FUNCTION_BLOCK DigitalOut
VAR_INPUT
END_VAR
VAR_OUTPUT
END_VAR
VAR
	DO_io  AT %Q*: BOOL;
	timerOn : TON;
	timerOff : TON;
	onActive : BOOL;
	offActive : BOOL;
	Do_in: BOOL;
	ActualCycle : UDINT;
	fbGetCurrTask : GETCURTASKINDEX;
	NextOn: UDINT;
	NextOff :UDINT;
	fifo : FB_Fifo;
	NextOnOff : ST_streamOutputs;
	init: BOOL;
END_VAR


IF init THEN
	init := FALSE;
	fifo.M_init();
	NextOnoff.cycleNo := 0;
END_IF



ActualCycle := TwinCAT_SystemInfoVarList._TaskInfo[1].CycleCount;
fifo();



IF fifo.bDataInBuffer AND NextOnOff.cycleNo = 0 THEN
	NextOnOff := fifo.M_RemoveEntry();
END_IF


IF ActualCycle = NextOnOff.cycleNo THEN
	NextOnOff.cycleNo := 0;
	DO_io := nextonoff.on;
END_IF

{attribute 'TcRpcEnable'}
METHOD M_OffWithDelay : BOOL
VAR_INPUT
	cycleNo : INT;
END_VAR

VAR

END_VAR



NextOff := ActualCycle + cycleNo + FIFOaxis.NrOccupiedLines;


fifo.M_AddEntry(NextOff, FALSE);
END_METHOD

{attribute 'TcRpcEnable'}
METHOD M_OnWithDelay : BOOL
VAR_INPUT
	cycleNo : INT;
END_VAR

VAR

END_VAR


NextOn := ActualCycle + cycleNo + FIFOaxis.NrOccupiedLines;

fifo.M_AddEntry(NextOn, TRUE);
END_METHOD

END_FUNCTION_BLOCK

(* stored: Version 1.1.0.1, ProductVersion 3.1.4024.9
   POU DigitalOut: Id {fda46c6a-9c06-4569-ac86-951c221ad104}, SpecialFunc None
   Method M_OffWithDelay: Id {d9c3e10c-c906-4b2e-bdb8-3cfbc05c03b4}
   Method M_OnWithDelay: Id {4adbf21e-db70-46e3-aa63-3283b18def19} *)
